FUNCTION_BLOCK PUBLIC FB_ElementForkInterface IMPLEMENTS ITF_PB_ElementForkInterface

VAR
	_ForkStatus			: ST_ForkState;
	_ForkRequest			: ST_ForkRequest;
END_VAR

//_ForkStatus := ForkStatus;
//ForkRequest := _ForkRequest;

PROPERTY P_ForkRequest : ST_ForkRequest
GET
P_ForkRequest := _ForkRequest;
END_GET
SET
_ForkRequest := P_ForkRequest;
END_SET
END_PROPERTY

PROPERTY P_ForkStatus : ST_ForkState
GET
P_ForkStatus := _ForkStatus;
END_GET
SET
_ForkStatus := P_ForkStatus;
END_SET
END_PROPERTY

END_FUNCTION_BLOCK

(* stored: Version 1.1.0.1, ProductVersion 3.1.4024.9
   POU FB_ElementForkInterface: Id {05b3492b-544d-4232-bcdb-6b4566b9ba61}, SpecialFunc None
   Property P_ForkRequest: Id {45ae1024-f5b0-46be-88f4-2a37dd8a02e5}
   Get Get: Id {3d4ed188-ef0c-4517-9731-c0bf353a4728}
   Set Set: Id {584339eb-4216-462d-a608-19ba6ce28414}
   Property P_ForkStatus: Id {d53712e3-55cc-4e4b-a060-c41d97379972}
   Get Get: Id {0f0a8fb6-b568-4374-8c11-bacb680e7cb9}
   Set Set: Id {ec21fb32-a24f-4f08-9954-955b6b34e82d} *)
